{attribute 'qualified_only'}
VAR_GLOBAL
END_VAR

(* stored: Version 1.1.0.1, ProductVersion 3.1.4022.7
   GVL GVL_05_Manual_Servo_Motor_Robot: Id {293719a6-abf4-4f3e-945c-357b457ada44} *)
